// TIA Portal V20 export
TYPE "OPC_SystStatus_Ack"
// stored: Namespace ProductionLine
   STRUCT
      AckSeq : Int;
   END_STRUCT;
END_TYPE
